{attribute 'GeneratedUsingTerminal: EL9576-0000-0016'}
{attribute addProperty BoxType "EL9576-0000-0016"}
{attribute addProperty Id "EtcSlaveTerminalBaseBCT_InputsAT %I*BCT_Inputs_28C1780C15WcStateAT %I*WcState_9091E0EB2InfoDataAT %I*InfoData_32EB74EA10"}
{attribute addProperty CRC "511639145"}
{attribute addProperty Size "27"}
TYPE EL9576_1E7EFE69 EXTENDS EtcSlaveTerminalBase :
STRUCT
	{attribute addProperty Name "BCT_Inputs"}
	BCT_Inputs : BCT_Inputs_28C1780C;
	{attribute addProperty Name "WcState"}
	WcState : WcState_9091E0EB;
	{attribute addProperty Name "InfoData"}
	InfoData : InfoData_32EB74EA;
END_STRUCT
END_TYPE

(* stored: Version 1.2.0.0, ProductVersion 3.1.4024.9
   DUT EL9576_1E7EFE69: Id {0a1b92f9-53e0-4968-9f39-d37bbe38cd1f} *)
